(* CoDeSys 2.3.9.41 project: Пульт управления А-М.pro *)
(* Libraries: STANDARD.LIB 4.10.05 11:14:46, IECSFC.LIB 13.4.06 15:51:28, SYSLIBTIME.LIB 20.2.06 12:31:16, SYSTASKINFO.LIB 20.2.06 12:31:38, ANALYZATION.LIB 5.10.99 09:05:06, SysLibFile.lib 20.2.06 12:31:10, SYSLIBCALLBACK.LIB 20.2.06 12:31:08 *)

(* PLC configuration (modules and I/O channels)
pumpButton AT %IX0.0 [BitInput]
workButton AT %IX0.1 [BitInput]
AT %IX0.2 [BitInput]
AT %IX0.3 [BitInput]
AT %IX0.4 [BitInput]
AT %IX0.5 [BitInput]
Discrete output 4 bit [ID101] node 1, in %IB1 out %QB1 {PinCount = 4; SafeValueBool = FALSE; SafeValueBool = FALSE; SafeValueBool = FALSE; SafeValueBool = FALSE; Visibility = No}
  AT %QX1.0 [BitOutput]
  AT %QX1.1 [BitOutput]
  AT %QX1.2 [BitOutput]
  AT %QX1.3 [BitOutput]
Special output [ID104] node 2, in %IB2 out %QB2 {Visibility = No; PinCount = 1}
  AT %QX2.0 [BitOutput] Special output
Unifed signal sensor [ID700] node 3, in %IB3 out %QB3 {Type_of_sensor700 = R0_5000; measure_interval = 0.8; ainlow = 4; ainhigh = 20; first_cor_point = 0; first_delta = 0; second_cor_point = 0; second_delta = 0; third_cor_point = 0; third_delta = 0; Visibility = No}
  AT %ID3.0 [FloatInput] Value
  AT %IW3.1 [WordInput] Circular time
  Analog Input [ID107] node 0, in %IB3.0 out %QB3.0
Unifed signal sensor [ID700] node 4, in %IB4 out %QB4 {Type_of_sensor700 = R0_5000; measure_interval = 0.8; ainlow = 0; ainhigh = 25000; first_cor_point = 0; first_delta = 0; second_cor_point = 0; second_delta = 0; third_cor_point = 0; third_delta = 0; Visibility = No}
  AT %ID4.0 [FloatInput] Value
  AT %IW4.1 [WordInput] Circular time
  Analog Input [ID107] node 0, in %IB4.0 out %QB4.0
Unifed signal sensor [ID700] node 5, in %IB5 out %QB5 {Type_of_sensor700 = IT_4_20; measure_interval = 0.8; ainlow = 0; ainhigh = 25000; first_cor_point = 0; first_delta = 0; second_cor_point = 0; second_delta = 0; third_cor_point = 0; third_delta = 0; Visibility = No}
  CurrentPressureIn AT %ID5.0 [FloatInput] Value
  AT %IW5.1 [WordInput] Circular time
  Analog Input [ID107] node 0, in %IB5.0 out %QB5.0
Unifed signal sensor [ID700] node 6, in %IB6 out %QB6 {Type_of_sensor700 = IT_4_20; measure_interval = 0.8; ainlow = 0; ainhigh = 25000; first_cor_point = 0; first_delta = 0; second_cor_point = 0; second_delta = 0; third_cor_point = 0; third_delta = 0; Visibility = No}
  AT %ID6.0 [FloatInput] Value
  AT %IW6.1 [WordInput] Circular time
  Analog Input [ID107] node 0, in %IB6.0 out %QB6.0
Analog output [ID106] node 7, in %IB7 out %QB7 {DAC_Type = Voltage 0-10 B; Analog_offset_correction = 0; Analog_full_range_correction = 0; SafeValueFloat = 0; Visibility = No}
  AT %QD7.0 [FloatOutput] Value
Analog output [ID106] node 8, in %IB8 out %QB8 {DAC_Type = Voltage 0-10 B; Analog_offset_correction = 0; Analog_full_range_correction = 0; SafeValueFloat = 0; Visibility = No}
  AT %QD8.0 [FloatOutput] Value
AT %QD9.0 [DWordOutput] Last address
AT %QW9.1 [WordOutput] Last error
RS-485-1 [COM1_USART] node 0, in %IB9.0 out %QB9.0 {CommunicationSpeed = 9600; Parity = NO PARITY CHECK; BitLength = 8 bits; StopLength = One stop bit; InterfaceType = RS485; FrameOriented = RTU; Timeout = 0; Visibility = No}
Universal Modbus device [ID2000] node 1, in %IB9.1 out %QB9.1 {ModuleIP = 10:1:1:239; ServiceTimeout = 150; TCPport = 502; NetMode = Serial; ModuleSlaveAddress = 1; RequestType = By poll time; PeriodOfService = 100; Visibility = No; RepeatCounter = 0; ByteSequence = Trace_mode}
  AT %QB9.1.0 [ComChannel] Command (0xff - Start)
OffIn AT %IW9.1.0.0 [WordInput]
currentPressure AT %QW9.1.1.0 [WordOutput]
OnIn AT %IW9.1.2.0 [WordInput]
PUMP_STATUS AT %QW9.1.3.0 [WordOutput]
OnOut AT %QW9.1.4.0 [WordOutput]
OffOut AT %QW9.1.5.0 [WordOutput]
AT %QB9.2.0 [ComChannel] Command (0xff - Start)
PUMP_ON_COMMAND AT %QW9.2.1.0 [WordOutput]
coming AT %IW9.2.2.0 [WordInput]
outGoing AT %QW9.2.3.0 [WordOutput]
plcStatus AT %IW9.2.4.0 [WordInput]
*)

(* POU PLC_PRG, ST *)
PROGRAM PLC_PRG
	VAR
	TURN_ON:BOOL:=FALSE;
	initial:BOOL:=TRUE;
	fileName:DWORD;
	initTon:TON;(*Таймер инициализации*)

	pressure : ARRAY[1..2] OF INT; (*Уставки давления 1 Верх , 2 низ*)
	checkValue:INT:=0;
	TURN_OFF_DELAY:TOF; (*Задержка отключения насоса при быстром изменении показания давления на нижней уставке*)
	checkPD:BOOL:=TRUE; (*Включение проверки наличия датчика*)
	connectTon:TON; (*Таймер отслеживания наличия сети*)

	(*Данные для SCADA системы*)
	SCADA_OFF:REAL;
	SCADA_ON:REAL;
	SCADA_ENABLE:BOOL:=FALSE;
	SCADA_STATUS:INT;
	SCADA_PRESSURE:REAL;
END_VAR
TURN_OFF_DELAY(PT:=T#50s);
initTon(PT:=T#20s);
connectTon(PT:=T#3m);

CurrentPressure:=REAL_TO_WORD(CurrentPressureIn* 0.98692);
SCADA_PRESSURE:=CurrentPressure;

(*Инициализация параметров нижнего и верхнего порога при запуске ПЛК*)
IF initial THEN
	fileName:=SysFileOpen('pressure.txt','r');
	SysFileRead(fileName,ADR(pressure),SIZEOF(pressure));
	OffOut:=pressure[1];
	OnOut:=pressure[2];
	outGoing:=checkValue;
	initial:=FALSE;
	initTon.IN:=NOT initial;
	SysFileClose(fileName);
END_IF

(*Поправка введенных данных с пульта*)
IF OnIn<OffIn  AND OnIn<>OffIn AND OffIn<>0 AND OnIn <>0  AND OnIn>0 AND OffIn>0 THEN
	IF OnOut<>OnIn THEN
		OnOut:=OnIn;
	END_IF;
	IF OffOut <> OffIn THEN
		OffOut:=OffIn;
	END_IF
END_IF;

(*Записать изменения в файл*)
IF pressure[1]<>OffOut  OR pressure[2] <> OnOut THEN
	pressure[1]:=OffOut; pressure[2]:=OnOut;
	SCADA_OFF:=pressure[1];
	SCADA_ON:=pressure[2];
	fileName:=SysFileOpen('pressure.txt','w');
	SysFileWrite(fileName,ADR(pressure),SIZEOF(pressure));
	SysFileClose(fileName);
END_IF;

(*включение при достижении нижнего порога*)
IF (CurrentPressure <= OnOut OR (SCADA_ENABLE AND SCADA_PRESSURE<=SCADA_ON)) AND initTon.Q THEN
	TURN_OFF_DELAY.IN:=TRUE;
END_IF
(*отключение при достижении верхнего порога*)
IF (CurrentPressure >= OffOut  OR (SCADA_ENABLE AND SCADA_PRESSURE>=SCADA_OFF) AND initTon.Q)  THEN
	TURN_OFF_DELAY.IN:=FALSE;
END_IF

TURN_ON:=TURN_OFF_DELAY.Q;

(*Проверка Наличия связи между контроллерами*)
connectTon.IN:=TRUE;
IF plcStatus=outGoing  THEN
	IF outGoing >24 THEN
		outGoing:=0;
	ELSE
		outGoing:=outGoing+1;
	END_IF
	PUMP_STATUS:=0;
	connectTon.IN:=FALSE;
ELSIF connectTon.Q THEN
	PUMP_STATUS:=6;
END_IF;



(*Проверка наличия датчика*)
IF checkPD AND CurrentPressureIn<0 THEN
	PUMP_STATUS:=7;
	PUMP_ON_COMMAND:=7;
	SCADA_ENABLE:=FALSE;
(*Уведомление об аварийной остановке*)
ELSIF NOT workButton THEN
	SCADA_ENABLE:=FALSE;
	PUMP_STATUS:=5;
	PUMP_ON_COMMAND:=5;
ELSIF PUMP_STATUS =6 THEN
	PUMP_STATUS:=6;
(*Включение Оператором со скады системы*)
ELSIF coming=15 THEN
	PUMP_STATUS:=1;
(*Включение  при достижении нижнего порога*)
ELSIF TURN_ON THEN
	PUMP_STATUS:=3;
	PUMP_ON_COMMAND:=3;
(*Включение при нажатии кнопки на первом пине*)
ELSIF pumpButton   THEN
	SCADA_ENABLE:=FALSE;
	PUMP_STATUS:=4;
	PUMP_ON_COMMAND:=4;
(*Включение с кургазака*)
ELSIF (coming=2 AND PUMP_ON_COMMAND=0) THEN
	SCADA_ENABLE:=FALSE;
	PUMP_STATUS:=2;
	PUMP_ON_COMMAND:=0;
(*Отключение насоса*)
ELSE
	PUMP_STATUS:=0;
	PUMP_ON_COMMAND:=0;
END_IF

SCADA_STATUS:=PUMP_STATUS;
END_PROGRAM
